TYPE ST_Places_Inputs_1 :
STRUCT
END_STRUCT
END_TYPE

(* stored: Version 1.1.0.1, ProductVersion 3.1.4024.9
   DUT ST_Places_Inputs_1: Id {f1752029-6e73-4ff7-b2e9-1bbd108401ec} *)
